(* CODESYS project tcoio.library
   Company: Vortex.Library
   DefaultNamespace: TcoIo
   Version: 1.19.1.1780
   Placeholder: TcoIo
   Title: TcoIo

Project tree, tasks and I/O mapping:
  libraries: Tc2_EtherCAT, * (Beckhoff Automation GmbH); Tc2_Standard, * (Beckhoff Automation GmbH); Tc2_System, * (Beckhoff Automation GmbH); Tc3_Module, * (Beckhoff Automation GmbH); TcoCore, 0.6.0.913 (Vortex.Library)
  Diagnostics/
    EtherCAT/
      MasterDevice/
        Base/
          data type EtcMasterBase_62654B43
          data type SyncUnitsBase_AD6C35CE
          data type SyncUnitTaskBase_FCD3CBF3
          data type SyncUnitTasksBase_7C8711EB
        Messenger/
          function block DiagnosticsMessenger [ST]: FB_init
          function block DiagnosticsMessengers [ST]: FB_init
        SyncUnit/
          data type InfoData_8649EEEB
          interface ITcoSyncUnit: DataInvalid, DataValid, HasSomeIssue, State
          data type SyncUnitState
          data type SyncUnitTask_AB2F5079
          function block TcoSyncUnit [ST]: DataInvalid, DataValid, HasSomeIssue, State
        data type InfoData_84133AC9
        data type Inputs_A65FACA4
        interface ITcoEthercatMasterDevice: AllDataValid, DeviceHasSomeIssue, SomeDataInvalid, SomeSyncUnitHasSomeIssue, State
        data type Outputs_23C0ED1D
        function block TcoEthercatDiagnosticsTask [ST]: FB_init, OnAbort, OnDone, OnError, OnStart, Restore
        function block TcoEthercatMasterDevice [ST]: AllDataValid, DeviceHasSomeIssue, Diagnostics, FB_init, Restore, ServiceMode, SomeDataInvalid, SomeSyncUnitHasSomeIssue, State, SyncUnitHasSomeIssue, UpdateSyncUnitsStatus
        data type TcoEthercatMasterDeviceState
      SlaveDevice/
        Base/
          data type EtcSlaveBase_82538BE2
          data type EtcSlaveBoxBase_77A0E4A7
          data type EtcSlaveEndTerminalBase_866C7F0C
          data type EtcSlaveTerminalBase_947E5A46
        InfoData/
          data type InfoData_23CBA837
          data type InfoData_6F19DB2B
        Inputs/
          data type InputBase_8311D824
        Outputs/
          data type OutputBase_10CEE7DE
        WcState/
          data type WcState_0B2B16F9
          data type WcState_9091E0EB
      global variables TcoEthercat
  POUs/
    program MAIN [ST]
  SpecialPlcTypes/
    data type TcoAmsAddr
    data type TcoAmsNetId
*)

// Diagnostics/EtherCAT/MasterDevice/Base/EtcMasterBase_62654B43

TYPE EtcMasterBase_62654B43 :
STRUCT
END_STRUCT
END_TYPE

// Diagnostics/EtherCAT/MasterDevice/Base/SyncUnitsBase_AD6C35CE

TYPE SyncUnitsBase_AD6C35CE :
STRUCT
END_STRUCT
END_TYPE

// Diagnostics/EtherCAT/MasterDevice/Base/SyncUnitTaskBase_FCD3CBF3

TYPE SyncUnitTaskBase_FCD3CBF3 :
STRUCT
END_STRUCT
END_TYPE

// Diagnostics/EtherCAT/MasterDevice/Base/SyncUnitTasksBase_7C8711EB

TYPE SyncUnitTasksBase_7C8711EB :
STRUCT
END_STRUCT
END_TYPE

// Diagnostics/EtherCAT/MasterDevice/SyncUnit/InfoData_8649EEEB
{attribute 'GeneratedUsingTerminal: IODEVICETYPE_ETHERCATPROT'}
{attribute addProperty BoxType "IODEVICETYPE_ETHERCATPROT"}
{attribute addProperty Id "ObjectIdAT %I*DWORD4StateAT %I*UINT2SlaveCountAT %I*UINT2"}
{attribute addProperty CRC "2252992235"}
{attribute addProperty Size "8"}
TYPE InfoData_8649EEEB :
STRUCT
	{attribute addProperty Name "ObjectId"}
	ObjectId AT %I* : DWORD;
	{attribute addProperty Name "State"}
	State AT %I* : UINT;
	{attribute addProperty Name "SlaveCount"}
	SlaveCount AT %I* : UINT;
END_STRUCT
END_TYPE

// Diagnostics/EtherCAT/MasterDevice/SyncUnit/SyncUnitState
TYPE SyncUnitState :
STRUCT
	{attribute addProperty Name "At least one slave in 'INIT' state"}	
    AtLeastOneSlaveInInitState : BOOL;
	{attribute addProperty Name "At least one slave in 'PREOP' state"}	
    AtLeastOneSlaveInPreopState : BOOL;
	{attribute addProperty Name "At least one slave in 'BOOT' state"}	
    AtLeastOneSlaveInBootState : BOOL;
	{attribute addProperty Name "At least one slave in 'SAFEOP' state"}	
    AtLeastOneSlaveInSafeOpState : BOOL;
	{attribute addProperty Name "At least one slave in 'OP' state"}	
    AtLeastOneSlaveInOpState : BOOL;
	{attribute addProperty Name "At least one slave signals error"}	
    AtLeastOneSlaveSignalsError : BOOL;
	{attribute addProperty Name "Invalid vendorId, productCode... read"}	
    InvalidVendoridOrProductcodeRead : BOOL;
	{attribute addProperty Name "Initialization error occurred"}	
    InitializationErrorOccurred : BOOL;
	{attribute addProperty Name "At least one slave disabled"}	
    AtLeastOneSlaveDisabled : BOOL;
	{attribute addProperty Name "At least one slave not present"}	
    AtLeastOneSlaveNotPresent : BOOL;
	{attribute addProperty Name "At least one slave signals link error"}	
    AtLeastOneSlaveSignalsLinkError : BOOL;
	{attribute addProperty Name "At least one slave signals missing link"}	
    AtLeastOneSlaveSignalsMissingLink : BOOL;
	{attribute addProperty Name "At least one slave signals unexpected link"}	
    AtLeastOneSlaveSignalsUnexpectedLink : BOOL;	
END_STRUCT
END_TYPE

// Diagnostics/EtherCAT/MasterDevice/SyncUnit/SyncUnitTask_AB2F5079
{attribute 'GeneratedUsingTerminal: IODEVICETYPE_ETHERCATPROT'}
{attribute addProperty BoxType "IODEVICETYPE_ETHERCATPROT"}
{attribute addProperty Id "WcStateAT %I*WcState_0B2B16F91InfoDataAT %I*InfoData_8649EEEB8"}
{attribute addProperty CRC "2872004729"}
{attribute addProperty Size "9"}
TYPE SyncUnitTask_AB2F5079 EXTENDS SyncUnitTaskBase_FCD3CBF3 :
STRUCT
	{attribute addProperty Name "WcState"}
	WcState : WcState_0B2B16F9;
	{attribute addProperty Name "InfoData"}
	InfoData : InfoData_8649EEEB;
END_STRUCT
END_TYPE

// Diagnostics/EtherCAT/MasterDevice/InfoData_84133AC9
{attribute 'GeneratedUsingTerminal: IODEVICETYPE_ETHERCATPROT'}
{attribute addProperty BoxType "IODEVICETYPE_ETHERCATPROT"}
{attribute addProperty Id "ChangeCountAT %I*UINT2DevIdAT %I*UINT2AmsNetIdAT %I*AMSNETID6CfgSlaveCountAT %I*UINT2DcToTcTimeOffsetAT %I*LINT8DcToExtTimeOffsetAT %I*LINT8"}
{attribute addProperty CRC "3867959757"}
{attribute addProperty Size "28"}
TYPE InfoData_84133AC9 :
STRUCT
	{attribute addProperty Name "ChangeCount"}
	ChangeCount AT %I* : UINT;
	{attribute addProperty Name "DevId"}
	DevId AT %I* : UINT;
	{attribute addProperty Name "AmsNetId"}
	AmsNetId AT %I* : TcoAmsNetId;
	{attribute addProperty Name "CfgSlaveCount"}
	CfgSlaveCount AT %I* : UINT;
	{attribute addProperty Name "DcToTcTimeOffset"}
	DcToTcTimeOffset AT %I* : LINT;
	{attribute addProperty Name "DcToExtTimeOffset"}
	DcToExtTimeOffset AT %I* : LINT;
END_STRUCT
END_TYPE

// Diagnostics/EtherCAT/MasterDevice/Inputs_A65FACA4
{attribute 'GeneratedUsingTerminal: IODEVICETYPE_ETHERCATPROT'}
{attribute addProperty BoxType "IODEVICETYPE_ETHERCATPROT"}
{attribute addProperty Id "SlaveCountAT %I*UINT2DevStateAT %I*UINT2Frm0StateAT %I*UINT2Frm0WcStateAT %I*UINT2Frm0InputToggleAT %I*UINT2"}
{attribute addProperty CRC "2791287972"}
{attribute addProperty Size "10"}
TYPE Inputs_A65FACA4 :
STRUCT
	{attribute addProperty Name "SlaveCount"}
	SlaveCount AT %I* : UINT;
	{attribute addProperty Name "DevState"}
	DevState AT %I* : UINT;
	{attribute addProperty Name "Frm0State"}
	Frm0State AT %I* : UINT;
	{attribute addProperty Name "Frm0WcState"}
	Frm0WcState AT %I* : UINT;
	{attribute addProperty Name "Frm0InputToggle"}
	Frm0InputToggle AT %I* : UINT;
END_STRUCT
END_TYPE

// Diagnostics/EtherCAT/MasterDevice/Outputs_23C0ED1D
{attribute 'GeneratedUsingTerminal: IODEVICETYPE_ETHERCATPROT'}
{attribute addProperty BoxType "IODEVICETYPE_ETHERCATPROT"}
{attribute addProperty Id "DevCtrlAT %Q*UINT2Frm0CtrlAT %Q*UINT2Frm0WcCtrlAT %Q*UINT2"}
{attribute addProperty CRC "599846173"}
{attribute addProperty Size "6"}
TYPE Outputs_23C0ED1D :
STRUCT
	{attribute addProperty Name "DevCtrl"}
	DevCtrl AT %Q* : UINT;
	{attribute addProperty Name "Frm0Ctrl"}
	Frm0Ctrl AT %Q* : UINT;
	{attribute addProperty Name "Frm0WcCtrl"}
	Frm0WcCtrl AT %Q* : UINT;
END_STRUCT
END_TYPE

// Diagnostics/EtherCAT/MasterDevice/TcoEthercatMasterDeviceState
TYPE TcoEthercatMasterDeviceState : STRUCT
	{attribute addProperty Name "Link error"}	
    LinkError : BOOL;
	{attribute addProperty Name "I/O locked after link error (I/O reset required)"}	
    IOLockedAfterLinkError : BOOL;
	{attribute addProperty Name "Link error (redundancy adapter)"}	
    LinkErrorRedundancyAdapter : BOOL;
	{attribute addProperty Name "Missing one frame (redundancy mode)"}	
    MissingOneFrame : BOOL;
	{attribute addProperty Name "Out of send resources (I/O reset required)"}	
    OutOfSendResources : BOOL;
	{attribute addProperty Name "Watchdog triggered"}	
    WatchdogTriggered : BOOL;
	{attribute addProperty Name "Ethernet driver (miniport) not found"}	
    EthernetDriverNotFound : BOOL;
	{attribute addProperty Name "I/O reset active"}	
    IOResetActive : BOOL;
	{attribute addProperty Name "At least one slave in 'INIT' state"}	
    AtLeastOneDeviceInInitState : BOOL;
	{attribute addProperty Name "At least one slave in 'PREOP' state"}	
    AtLeastOneDeviceInPreOpState : BOOL;
	{attribute addProperty Name "At least one slave in 'SAFEOP' state"}	
    AtLeastOneDeviceInSafeOpState : BOOL;
	{attribute addProperty Name "At least one device indicates an error state"}	
    AtLeastOneDeviceIndicatesAnErrorState : BOOL;
	{attribute addProperty Name "DC not in sync"}	
    DcNotInSync : BOOL;
END_STRUCT
END_TYPE

// Diagnostics/EtherCAT/SlaveDevice/Base/EtcSlaveBase_82538BE2

TYPE EtcSlaveBase_82538BE2 :
STRUCT
END_STRUCT
END_TYPE

// Diagnostics/EtherCAT/SlaveDevice/Base/EtcSlaveBoxBase_77A0E4A7

{attribute clr[Container(Layout.Stack)]}
{attribute clr[Group(Layout.GroupBox)]}
{attribute addProperty PreviousPort "Unknown"}
{attribute addProperty SyncUnit "Unknown"}
TYPE EtcSlaveBoxBase_77A0E4A7 EXTENDS EtcSlaveBase_82538BE2 :
STRUCT
END_STRUCT
END_TYPE

// Diagnostics/EtherCAT/SlaveDevice/Base/EtcSlaveEndTerminalBase_866C7F0C

{attribute clr[Container(Layout.Stack)]}
{attribute clr[Group(Layout.GroupBox)]}
{attribute addProperty PreviousPort "Unknown"}
{attribute addProperty SyncUnit "Unknown"}
TYPE EtcSlaveEndTerminalBase_866C7F0C EXTENDS TcoIo.EtcSlaveBase_82538BE2 :
STRUCT
END_STRUCT
END_TYPE

// Diagnostics/EtherCAT/SlaveDevice/Base/EtcSlaveTerminalBase_947E5A46

{attribute clr[Container(Layout.Stack)]}
{attribute clr[Group(Layout.GroupBox)]}
{attribute addProperty PreviousPort "Unknown"}
{attribute addProperty SyncUnit "Unknown"}
TYPE EtcSlaveTerminalBase_947E5A46 EXTENDS EtcSlaveBase_82538BE2 :
STRUCT
END_STRUCT
END_TYPE

// Diagnostics/EtherCAT/SlaveDevice/InfoData/InfoData_23CBA837
{attribute 'GeneratedUsingTerminal: EL6002-0000-0019'}
{attribute addProperty BoxType "EL6002-0000-0019"}
{attribute addProperty Id "AdsAddrAT %I*TcoIo.TcoAmsAddr0StateAT %I*UINT2"}
{attribute addProperty CRC "600549431"}
{attribute addProperty Size "2"}
TYPE InfoData_23CBA837 :
STRUCT
	{attribute addProperty Name "AdsAddr"}
	AdsAddr AT %I* : TcoAmsAddr;
	{attribute addProperty Name "State"}
	State AT %I* : UINT;
END_STRUCT
END_TYPE

// Diagnostics/EtherCAT/SlaveDevice/InfoData/InfoData_6F19DB2B
{attribute 'GeneratedUsingTerminal: EL1809-0000-0018'}
{attribute addProperty BoxType "EL1809-0000-0018"}
{attribute addProperty Id "StateAT %I*UINT2"}
{attribute addProperty CRC "1863965483"}
{attribute addProperty Size "2"}
TYPE InfoData_6F19DB2B :
STRUCT
	{attribute addProperty Name "State"}
	State AT %I* : UINT;
END_STRUCT
END_TYPE

// Diagnostics/EtherCAT/SlaveDevice/Inputs/InputBase_8311D824

TYPE InputBase_8311D824 :
STRUCT
END_STRUCT
END_TYPE

// Diagnostics/EtherCAT/SlaveDevice/Outputs/OutputBase_10CEE7DE

TYPE OutputBase_10CEE7DE :
STRUCT
END_STRUCT
END_TYPE

// Diagnostics/EtherCAT/SlaveDevice/WcState/WcState_0B2B16F9
{attribute 'GeneratedUsingTerminal: EL2809-0000-0018'}
{attribute addProperty BoxType "EL2809-0000-0018"}
{attribute addProperty Id "WcStateAT %I*BOOL1"}
{attribute addProperty CRC "187373305"}
{attribute addProperty Size "1"}
TYPE WcState_0B2B16F9 :
STRUCT
	{attribute addProperty Name "WcState"}
	WcState AT %I* : BOOL;
END_STRUCT
END_TYPE

// Diagnostics/EtherCAT/SlaveDevice/WcState/WcState_9091E0EB
{attribute 'GeneratedUsingTerminal: EL6002-0000-0019'}
{attribute addProperty BoxType "EL6002-0000-0019"}
{attribute addProperty Id "WcStateAT %I*BOOL1InputToggleAT %I*BOOL1"}
{attribute addProperty CRC "2425479403"}
{attribute addProperty Size "2"}
TYPE WcState_9091E0EB :
STRUCT
	{attribute addProperty Name "WcState"}
	WcState AT %I* : BOOL;
	{attribute addProperty Name "InputToggle"}
	InputToggle AT %I* : BOOL;
END_STRUCT
END_TYPE

// SpecialPlcTypes/TcoAmsAddr
TYPE TcoAmsAddr :
	STRUCT
		netId : ARRAY [0..5] OF BYTE;
		port : WORD;
	END_STRUCT
END_TYPE

// SpecialPlcTypes/TcoAmsNetId
TYPE TcoAmsNetId  :
	STRUCT
		netId : ARRAY [0..5] OF BYTE;
	END_STRUCT
END_TYPE

// Diagnostics/EtherCAT/TcoEthercat
{attribute 'qualified_only'}
VAR_GLOBAL CONSTANT
    C_MaxSyncUnits : UINT := 10;
	C_MAX_LOCAL_ERROR_MESSAGES : UINT := 3;	
END_VAR

// Diagnostics/EtherCAT/MasterDevice/Messenger/DiagnosticsMessenger
FUNCTION_BLOCK DiagnosticsMessenger EXTENDS TcoCore.TcoMessenger

{attribute 'hide'}
METHOD FB_init : BOOL
VAR_INPUT
	bInitRetains : BOOL; // if TRUE, the retain variables are initialized (warm start / cold start)
	bInCopyCode : BOOL;  // if TRUE, the instance afterwards gets moved into the copy code (online change)
	ParentObject : ITcoObject;
END_VAR
END_METHOD

END_FUNCTION_BLOCK

// Diagnostics/EtherCAT/MasterDevice/Messenger/DiagnosticsMessengers
FUNCTION_BLOCK DiagnosticsMessengers EXTENDS TcoCore.TcoObject
VAR
	Messengers : ARRAY [0..2] OF DiagnosticsMessenger(THIS^);
END_VAR

{attribute 'hide'}
METHOD FB_init : BOOL
VAR_INPUT
	bInitRetains : BOOL; // if TRUE, the retain variables are initialized (warm start / cold start)
	bInCopyCode : BOOL;  // if TRUE, the instance afterwards gets moved into the copy code (online change)
	ParentObject : ITcoObject;	
END_VAR
Messengers[0].FB_init(bInitRetains,bInCopyCode,ParentObject);
Messengers[1].FB_init(bInitRetains,bInCopyCode,ParentObject);
Messengers[2].FB_init(bInitRetains,bInCopyCode,ParentObject);
END_METHOD

END_FUNCTION_BLOCK

// Diagnostics/EtherCAT/MasterDevice/SyncUnit/ITcoSyncUnit
INTERFACE ITcoSyncUnit

PROPERTY DataInvalid : BOOL
GET
END_GET
END_PROPERTY

PROPERTY DataValid : BOOL
GET
END_GET
END_PROPERTY

PROPERTY HasSomeIssue : BOOL
GET
END_GET
END_PROPERTY

PROPERTY State : SyncUnitState
GET
END_GET
END_PROPERTY

END_INTERFACE

// Diagnostics/EtherCAT/MasterDevice/SyncUnit/TcoSyncUnit
FUNCTION_BLOCK TcoSyncUnit EXTENDS TcoCore.TcoObject IMPLEMENTS ITcoSyncUnit
VAR
    {attribute addProperty Name "WcState"}
    WcState : WcState_0B2B16F9;
    {attribute addProperty Name "InfoData"}
    InfoData : InfoData_8649EEEB;
    {attribute addProperty Name "Status"}
    _State : SyncUnitState;
    {attribute 'hide'}
    _hasSomeIssue : BOOL;
    {attribute 'hide'}
    _dataValid : BOOL;
    {attribute 'hide'}
    _dataInvalid : BOOL;
END_VAR

PROPERTY DataInvalid : BOOL
GET
_dataInvalid := WcState.WcState;
DataInvalid := _dataInvalid;
END_GET
END_PROPERTY

PROPERTY DataValid : BOOL
GET
_dataValid := NOT WcState.WcState;
DataValid := _dataValid;
END_GET
END_PROPERTY

PROPERTY HasSomeIssue : BOOL
GET
VAR
	_syncUnitStatus : SyncUnitState;
END_VAR
_syncUnitStatus := State;

_hasSomeIssue := _syncUnitStatus.AtLeastOneSlaveInInitState OR
			_syncUnitStatus.AtLeastOneSlaveInPreopState OR
			_syncUnitStatus.AtLeastOneSlaveInBootState OR
			_syncUnitStatus.AtLeastOneSlaveInSafeOpState OR
			_syncUnitStatus.AtLeastOneSlaveSignalsError OR
			_syncUnitStatus.InvalidVendoridOrProductcodeRead OR
			_syncUnitStatus.InitializationErrorOccurred OR
			_syncUnitStatus.AtLeastOneSlaveNotPresent OR
			_syncUnitStatus.AtLeastOneSlaveSignalsLinkError OR
			_syncUnitStatus.AtLeastOneSlaveSignalsMissingLink OR
			_syncUnitStatus.AtLeastOneSlaveSignalsUnexpectedLink;
	
HasSomeIssue := _hasSomeIssue;
END_GET
END_PROPERTY

PROPERTY State : SyncUnitState
GET
_State.AtLeastOneSlaveInInitState := InfoData.State.0 AND NOT InfoData.State.1;
_State.AtLeastOneSlaveInPreopState := InfoData.State.0 AND InfoData.State.1;
_State.AtLeastOneSlaveInBootState := InfoData.State.0 AND InfoData.State.1;
_State.AtLeastOneSlaveInSafeOpState := InfoData.State.2;
_State.AtLeastOneSlaveInOpState := InfoData.State.3;
_State.AtLeastOneSlaveSignalsError := InfoData.State.4;
_State.InvalidVendoridOrProductcodeRead := InfoData.State.5;
_State.InitializationErrorOccurred := InfoData.State.6;
_State.AtLeastOneSlaveDisabled := InfoData.State.7;
_State.AtLeastOneSlaveNotPresent := InfoData.State.8;
_State.AtLeastOneSlaveSignalsLinkError := InfoData.State.9;
_State.AtLeastOneSlaveSignalsMissingLink := InfoData.State.10;
_State.AtLeastOneSlaveSignalsUnexpectedLink := InfoData.State.11;

State := _State;
END_GET
END_PROPERTY

END_FUNCTION_BLOCK

// Diagnostics/EtherCAT/MasterDevice/ITcoEthercatMasterDevice
INTERFACE ITcoEthercatMasterDevice

PROPERTY AllDataValid : BOOL
GET
END_GET
END_PROPERTY

PROPERTY DeviceHasSomeIssue : BOOL
GET
END_GET
END_PROPERTY

PROPERTY SomeDataInvalid : BOOL
GET
END_GET
END_PROPERTY

PROPERTY SomeSyncUnitHasSomeIssue : BOOL
GET
END_GET
END_PROPERTY

PROPERTY State : TcoEthercatMasterDeviceState
GET
END_GET
END_PROPERTY

END_INTERFACE

// Diagnostics/EtherCAT/MasterDevice/TcoEthercatDiagnosticsTask
FUNCTION_BLOCK TcoEthercatDiagnosticsTask EXTENDS TcoCore.TcoTask
VAR_INPUT
	inNetId : Tc2_System.T_AmsNetID;
END_VAR
VAR
    _EcGetAllSlaveStates 	: Tc2_EtherCAT.FB_EcGetAllSlaveStates;
    _EcGetConfSlaves 		: Tc2_EtherCAT.FB_EcGetConfSlaves;
	_updateDiagnosticsState : TcoCore.TcoState(THIS^,TcoCore.eRestoreMode.None);

	_SlaveStatesCount      		: UINT;
    _ConfigSlavesCount     		: UINT;
    _SlaveStateBuffer      		: ARRAY[0..EC_MAX_SLAVES] OF Tc2_EtherCAT.ST_EcSlaveState;
    _SlaveConfigDataBuffer 		: ARRAY[0..EC_MAX_SLAVES] OF Tc2_EtherCAT.ST_EcSlaveConfigData;

	_i	:	UINT;

	_name : STRING;
	_type : STRING;
	_state : STRING;
	
	_DiagnosticsMessengers		: DiagnosticsMessengers(THIS^);
	_DiagnosticsMessengerIndex	: UINT;	
END_VAR
VAR_OUTPUT
	outDiagnosticsAvailable : BOOL;
END_VAR

IF Execute() THEN
	IF _updateDiagnosticsState.State = 10 THEN
		outDiagnosticsAvailable := FALSE;
		_EcGetAllSlaveStates(bExecute := FALSE);
		_EcGetConfSlaves(bExecute := FALSE);
	
		IF NOT _EcGetAllSlaveStates.bBusy AND NOT _EcGetAllSlaveStates.bError AND NOT _EcGetConfSlaves.bBusy AND NOT _EcGetConfSlaves.bError THEN
			_updateDiagnosticsState.ChangeState(_updateDiagnosticsState._State + 10);
		END_IF
	END_IF
	
	IF _updateDiagnosticsState.State = 20 THEN
		_EcGetAllSlaveStates(sNetId := inNetId,
			pStateBuf := ADR(_SlaveStateBuffer),
			cbBufLen := SIZEOF(_SlaveStateBuffer),
			bExecute := TRUE,
			tTimeout :=,
			bBusy =>,
			bError =>,
			nErrId =>,
			nSlaves => _SlaveStatesCount);
	
		IF _EcGetAllSlaveStates.bBusy THEN
			_updateDiagnosticsState.ChangeState(_updateDiagnosticsState._State + 10);
		END_IF
	END_IF
	
	IF _updateDiagnosticsState.State = 30 THEN
		_EcGetAllSlaveStates(sNetId := inNetId,
			pStateBuf := ADR(_SlaveStateBuffer),
			cbBufLen := SIZEOF(_SlaveStateBuffer),
			bExecute := FALSE,
			tTimeout :=,
			bBusy =>,
			bError =>,
			nErrId =>,
			nSlaves => _SlaveStatesCount);
	
		IF NOT _EcGetAllSlaveStates.bBusy AND NOT _EcGetAllSlaveStates.bError THEN
			_updateDiagnosticsState.ChangeState(_updateDiagnosticsState._State + 10);
		END_IF
	END_IF
	
	IF _updateDiagnosticsState.State = 40 THEN
		_EcGetConfSlaves(sNetId := inNetId,
			pArrEcConfSlaveInfo := ADR(_SlaveConfigDataBuffer),
			cbBufLen := SIZEOF(_SlaveConfigDataBuffer),
			bExecute := TRUE,
			tTimeout :=,
			bBusy =>,
			bError =>,
			nErrorId =>,
			nSlaves => _ConfigSlavesCount);
	
		IF _EcGetConfSlaves.bBusy THEN
			_updateDiagnosticsState.ChangeState(_updateDiagnosticsState._State + 10);
		END_IF
	END_IF
	
	IF _updateDiagnosticsState.State = 50 THEN
		_EcGetConfSlaves(sNetId := inNetId,
			pArrEcConfSlaveInfo := ADR(_SlaveConfigDataBuffer),
			cbBufLen := SIZEOF(_SlaveConfigDataBuffer),
			bExecute := FALSE,
			tTimeout :=,
			bBusy =>,
			bError =>,
			nErrorId =>,
			nSlaves => _ConfigSlavesCount);
	
		IF NOT _EcGetConfSlaves.bBusy AND NOT _EcGetConfSlaves.bError THEN
			_updateDiagnosticsState.ChangeState(_updateDiagnosticsState._State + 10);
		END_IF
	END_IF
	
	IF _updateDiagnosticsState.State = 60 THEN
		_EcGetAllSlaveStates(bExecute := FALSE);
		_EcGetConfSlaves(bExecute := FALSE);
	
		IF NOT _EcGetAllSlaveStates.bBusy AND NOT _EcGetAllSlaveStates.bError AND NOT _EcGetConfSlaves.bBusy AND NOT _EcGetConfSlaves.bError THEN
			_updateDiagnosticsState.ChangeState(_updateDiagnosticsState._State + 10);
		END_IF
	END_IF
	
	IF _updateDiagnosticsState.State = 70 THEN
		_DiagnosticsMessengerIndex := 0;
	    FOR _i := 0 TO _ConfigSlavesCount DO
			IF (_SlaveStateBuffer[_i].deviceState <> 8 OR _SlaveStateBuffer[_i].linkState <> 0) THEN
				IF _SlaveConfigDataBuffer[_i].sName <> '' THEN
					IF _DiagnosticsMessengerIndex <= 2 THEN
						outDiagnosticsAvailable := TRUE;
						_name := _SlaveConfigDataBuffer[_i].sName;
						_type := Tc2_EtherCAT.F_ConvProductCodeToString(_SlaveConfigDataBuffer[_i].stSlaveIdentity);
						_state :=  Tc2_EtherCAT.F_ConvSlaveStateToString(state := _SlaveStateBuffer[_i]);
						_DiagnosticsMessengers.Messengers[_DiagnosticsMessengerIndex].Build().AppendAny(_name).Append('[').AppendAny(_type).Append(']').Append( _state).As().AsError().Pin();
						_DiagnosticsMessengerIndex := _DiagnosticsMessengerIndex + 1;
					END_IF
				END_IF
			END_IF;
	    END_FOR

		_updateDiagnosticsState.ChangeState(_updateDiagnosticsState._State + 10);
	END_IF
	
	IF _updateDiagnosticsState.State = 80 THEN
		DoneWhen(TRUE);
	END_IF

	ThrowWhen(_EcGetAllSlaveStates.bError OR _EcGetConfSlaves.bError);
END_IF

METHOD FB_init : BOOL
VAR_INPUT
	bInitRetains : BOOL; // if TRUE, the retain variables are initialized (warm start / cold start)
	bInCopyCode : BOOL;  // if TRUE, the instance afterwards gets moved into the copy code (online change)
	ParentObject : TcoCore.ITcoObject;	
END_VAR
END_METHOD

(*~
	<docu>
		<summary>
			Executes when task is aborted.
		</summary>			
	</docu>	
~*)
METHOD PROTECTED OnAbort
_EcGetAllSlaveStates(bExecute := FALSE);
_EcGetConfSlaves(bExecute := FALSE);

_updateDiagnosticsState.Restore();
END_METHOD

(*~
	<docu>
		<summary>
			Executes when task reaches the ```Done``` state .
		</summary>			
	</docu>	
~*)
METHOD PROTECTED OnDone
_EcGetAllSlaveStates(bExecute := FALSE);
_EcGetConfSlaves(bExecute := FALSE);
END_METHOD

(*~
	<docu>
		<summary>
			Executes when task reaches the ```Error``` state.
			<para>
				Do not confuse with <see cref="PlcDocu.TcoCore.TcoTask.WhileError()"/>, that is called cyclically until '''Error''' state is left.
			</para>
		</summary>			
	</docu>	
~*)
METHOD PROTECTED OnError
IF _EcGetAllSlaveStates.bError THEN
	Messenger.Build().Append('Reading status of all EtherCAT slaves using "Tc2_EtherCAT.FB_EcGetAllSlaveStates" function block returns error. nErrId: ').AppendAny(_EcGetAllSlaveStates.nErrId).As().AsError();
ELSIF _EcGetConfSlaves.bError THEN
	Messenger.Build().Append('Reading status of configurateed EtherCAT slaves using "Tc2_EtherCAT.FB_EcGetConfSlaves" function block returns error. nErrorId: ').AppendAny(_EcGetConfSlaves.nErrorId).As().AsError();
END_IF
END_METHOD

METHOD PROTECTED OnStart
_EcGetAllSlaveStates(bExecute := FALSE);
_EcGetConfSlaves(bExecute := FALSE);

_updateDiagnosticsState.ChangeState(10);
END_METHOD

(*~
	<docu>
		<summary>
			Restores this instance to the Ready state. Can be called explicitly or from within one of the restore mechanisms.
			<para>
				See also <see cref="PlcDocu.TcoCore.TcoTask.AutoRestorable()"/>
			</para>
		</summary>			
	</docu>	
~*)
METHOD Restore : ITcoRestorable
THIS^._EcGetAllSlaveStates(bExecute := FALSE);
THIS^._EcGetConfSlaves(bExecute := FALSE);

THIS^._DiagnosticsMessengers.Messengers[0].Clear();
THIS^._DiagnosticsMessengers.Messengers[1].Clear();
THIS^._DiagnosticsMessengers.Messengers[2].Clear();

THIS^.outDiagnosticsAvailable := FALSE;
THIS^._updateDiagnosticsState.Restore();

SUPER^.Restore();
END_METHOD

END_FUNCTION_BLOCK

// Diagnostics/EtherCAT/MasterDevice/TcoEthercatMasterDevice
FUNCTION_BLOCK TcoEthercatMasterDevice EXTENDS TcoCore.TcoComponent IMPLEMENTS ITcoEthercatMasterDevice
VAR_INPUT
    Inputs   		:	Inputs_A65FACA4;
    InfoData		:	InfoData_84133AC9;
	SyncUnits		:	POINTER TO SyncUnitTask_AB2F5079;
	SyncUnitsSize	:	UINT;
END_VAR

VAR
    _someSyncUnitHasSomeIssue	: BOOL;
    _allDataValid          		: BOOL;
    _someDataInvalid       		: BOOL;
    _State                		: TcoEthercatMasterDeviceState;
    _NetId                 		: Tc2_System.T_AmsNetID;
    _DeviceHasSomeIssue    		: BOOL;
    _TcoEthercatDiagnosticsTask	: TcoEthercatDiagnosticsTask(THIS^);

    _InfoDataChangeCountPV 		: UINT;

	_numberOfSyncUnits			: UINT;

	{attribute addProperty Name "Acknowledge"}
	_acknowledge				:	TcoCore.TcoTask(THIS^);
	
	_DiagnosticsAvailable : BOOL;
END_VAR
VAR_OUTPUT
    Outputs  : Outputs_23C0ED1D;
END_VAR

UpdateSyncUnitsStatus(SyncUnits,SyncUnitsSize);
Diagnostics();

PROPERTY AllDataValid : BOOL
GET
AllDataValid := _allDataValid;
END_GET
END_PROPERTY

PROPERTY DeviceHasSomeIssue : BOOL
GET
_DeviceHasSomeIssue		:=	_State.LinkError							 	OR
							_State.IOLockedAfterLinkError 					OR
							_State.LinkErrorRedundancyAdapter	 			OR
							_State.MissingOneFrame 							OR
							_State.OutOfSendResources 						OR
							_State.WatchdogTriggered 						OR
							_State.EthernetDriverNotFound 					OR
							_State.IOResetActive 							OR
							_State.AtLeastOneDeviceInInitState 				OR
							_State.AtLeastOneDeviceInPreOpState 			OR
							_State.AtLeastOneDeviceInSafeOpState 			OR
							_State.AtLeastOneDeviceIndicatesAnErrorState 	OR
							_State.DcNotInSync 								;
							
DeviceHasSomeIssue := _DeviceHasSomeIssue;
END_GET
END_PROPERTY

METHOD Diagnostics
VAR
    _i : UINT;
END_VAR
_NetId := Tc2_System.F_CreateAmsNetId(InfoData.AmsNetId.netId);

_TcoEthercatDiagnosticsTask(inNetId := _NetId, outDiagnosticsAvailable => _DiagnosticsAvailable);

Service();

IF _acknowledge.Execute() THEN
	Restore();	
END_IF

IF (DeviceHasSomeIssue OR SomeSyncUnitHasSomeIssue OR SomeDataInvalid OR _InfoDataChangeCountPV <> InfoData.ChangeCount) (*OR _manualDiagnosticStart.Execute()*) THEN
	IF _TcoEthercatDiagnosticsTask.Ready THEN
		_InfoDataChangeCountPV := InfoData.ChangeCount;
		_TcoEthercatDiagnosticsTask.Invoke();
	END_IF
	IF _TcoEthercatDiagnosticsTask.Done AND NOT _DiagnosticsAvailable THEN
		_TcoEthercatDiagnosticsTask.Restore();
	END_IF;
END_IF
END_METHOD

METHOD FB_init : BOOL
VAR_INPUT
	bInitRetains : BOOL; // if TRUE, the retain variables are initialized (warm start / cold start)
	bInCopyCode : BOOL;  // if TRUE, the instance afterwards gets moved into the copy code (online change)
	ParentObject : TcoCore.ITcoObject;	
END_VAR
END_METHOD

(*~
	<docu>
		<summary>
			Restores this instance to the Ready state. Can be called explicitly or from within one of the restore mechanisms.	
		</summary>			
	</docu>	
~*)
METHOD  Restore : ITcoRestorable
THIS^.Messenger.Clear();
THIS^._DiagnosticsAvailable := FALSE;
THIS^._acknowledge.Restore();
THIS^._TcoEthercatDiagnosticsTask.Restore();
END_METHOD

(*~
	<docu>
		<summary>
		    Custom service (manual, maintenance) logic.
			This method must be implemented in derived class.
		</summary>			
	</docu>	
~*)
METHOD PROTECTED  ServiceMode
_acknowledge();
END_METHOD

PROPERTY SomeDataInvalid : BOOL
GET
SomeDataInvalid := _someDataInvalid;
END_GET
END_PROPERTY

PROPERTY SomeSyncUnitHasSomeIssue : BOOL
GET
SomeSyncUnitHasSomeIssue := _someSyncUnitHasSomeIssue;
END_GET
END_PROPERTY

PROPERTY State : TcoEthercatMasterDeviceState
GET
_State.LinkError							 	:= Inputs.DevState.0;
_State.IOLockedAfterLinkError 					:= Inputs.DevState.1;
_State.LinkErrorRedundancyAdapter	 			:= Inputs.DevState.2;
_State.MissingOneFrame 							:= Inputs.DevState.3;
_State.OutOfSendResources 						:= Inputs.DevState.4;
_State.WatchdogTriggered 						:= Inputs.DevState.5;
_State.EthernetDriverNotFound 					:= Inputs.DevState.6;
_State.IOResetActive 							:= Inputs.DevState.7;
_State.AtLeastOneDeviceInInitState 				:= Inputs.DevState.8;
_State.AtLeastOneDeviceInPreOpState 			:= Inputs.DevState.9;
_State.AtLeastOneDeviceInSafeOpState 			:= Inputs.DevState.10;
_State.AtLeastOneDeviceIndicatesAnErrorState 	:= Inputs.DevState.11;
_State.DcNotInSync 								:= Inputs.DevState.12;

State := _State;
END_GET
END_PROPERTY

METHOD SyncUnitHasSomeIssue : BOOL
VAR_INPUT
	inState : UINT;
END_VAR
VAR
	_state : SyncUnitState;
END_VAR
_state.AtLeastOneSlaveInInitState 				:=	inState.0 AND NOT	inState.1;
_state.AtLeastOneSlaveInPreopState 				:=	inState.0 AND 		inState.1;
_state.AtLeastOneSlaveInBootState 				:=	inState.0 AND		inState.1;
_state.AtLeastOneSlaveInSafeOpState 			:=	inState.2;
_state.AtLeastOneSlaveInOpState 				:=	inState.3;
_state.AtLeastOneSlaveSignalsError 				:=	inState.4;
_state.InvalidVendoridOrProductcodeRead 		:=	inState.5;
_state.InitializationErrorOccurred				:=	inState.6;
_state.AtLeastOneSlaveDisabled					:=	inState.7;
_state.AtLeastOneSlaveNotPresent				:=	inState.8;
_state.AtLeastOneSlaveSignalsLinkError			:=	inState.9;
_state.AtLeastOneSlaveSignalsMissingLink		:=	inState.10;
_state.AtLeastOneSlaveSignalsUnexpectedLink		:=	inState.11;

SyncUnitHasSomeIssue :=	_state.AtLeastOneSlaveInInitState OR
						_state.AtLeastOneSlaveInPreopState OR
						_state.AtLeastOneSlaveInBootState OR
						_state.AtLeastOneSlaveInSafeOpState OR
						_state.AtLeastOneSlaveSignalsError OR
						_state.InvalidVendoridOrProductcodeRead OR
						_state.InitializationErrorOccurred OR
						_state.AtLeastOneSlaveNotPresent OR
						_state.AtLeastOneSlaveSignalsLinkError OR
						_state.AtLeastOneSlaveSignalsMissingLink OR
						_state.AtLeastOneSlaveSignalsUnexpectedLink;
END_METHOD

METHOD UpdateSyncUnitsStatus
VAR_INPUT
	SyncUnits			:	POINTER TO SyncUnitTask_AB2F5079;
	SyncUnitsSize		:	UINT;
END_VAR
VAR
    _i					:	UINT;
	_pSyncUnit			:	POINTER TO SyncUnitTask_AB2F5079;
	_SyncUnit			:	SyncUnitTask_AB2F5079;
	_SyncUnitState		:	UINT;
END_VAR
_someSyncUnitHasSomeIssue := FALSE;
_allDataValid := TRUE;
_someDataInvalid := FALSE;

IF SyncUnits<>0 THEN
	_numberOfSyncUnits := SyncUnitsSize / SIZEOF(SyncUnitTask_AB2F5079);
	FOR _i := 0 TO _numberOfSyncUnits - 1 DO
		_pSyncUnit					:=	SyncUnits + _i * SIZEOF(SyncUnitTask_AB2F5079);
		_SyncUnit					:=	_pSyncUnit^;	
		_someSyncUnitHasSomeIssue 	:=	_someSyncUnitHasSomeIssue OR SyncUnitHasSomeIssue(_SyncUnit.InfoData.State);
		_allDataValid				:=	_allDataValid AND NOT _SyncUnit.WcState.WcState;
		_someDataInvalid			:=	_someDataInvalid OR _SyncUnit.WcState.WcState;
	END_FOR
END_IF
END_METHOD

END_FUNCTION_BLOCK

// POUs/MAIN
PROGRAM MAIN
VAR
END_VAR

END_PROGRAM
